# EPICS autosave request: iocBoot/sioc-li20-im02/sioc-li20-im02.req
file "facet2.req" AREA=LI20,POS=2452
file "facet2.req" AREA=LI20,POS=3163
